PROGRAM prgModbus
VAR
	PV1 :FB_SunSpec_PV_Inverter_T;
END_VAR

PV1(
	bEnable:= , 
	sIPAdress:= , 
	byUnitID_Inverter:= , 
	stDataSunSpec=> , 
	stDataEMPower_PV=> , 
	stDataEMCounter_PV=> , 
	diNrOfEM_OUT_PV=> );

END_PROGRAM

(* stored: Version 1.1.0.1, ProductVersion 3.1.4024.12
   POU prgModbus: Id {6a281e52-16a3-462b-9619-89d9dd6b702b}, SpecialFunc None *)
